FUNCTION_BLOCK MeasurementWidget
VAR_INPUT
    value : LREAL;
    actualStatus : STRING;
END_VAR
VAR_IN_OUT
    healthStatus : HealthStatus;
END_VAR
VAR_OUTPUT
    display : STRING;
    _formatString : FB_FormatString;
END_VAR
VAR
    name : STRING;
    actualStatusWidget : StatusWidget;
    format : STRING;
END_VAR

actualStatusWidget(text  := actualStatus,
                   color := HealthToColor(healthStatus));

IF healthStatus.good OR healthStatus.warning THEN
    _formatString(sFormat := format, 
                  arg1    := F_LREAL(value),
                  sOut    => display);
ELSE
    display := '';
END_IF

METHOD FB_init : BOOL
VAR_INPUT
	bInitRetains : BOOL; // if TRUE, the retain variables are initialized (warm start / cold start)
	bInCopyCode : BOOL;  // if TRUE, the instance afterwards gets moved into the copy code (online change)
    n : STRING;
    f : STRING;
END_VAR
name := n;
format := f;
END_METHOD

END_FUNCTION_BLOCK

(* stored: Version 1.1.0.1, ProductVersion 3.1.4018.2
   POU MeasurementWidget: Id {2fec0466-45e9-42aa-9920-0e9c2cbcfe65}, SpecialFunc None
   Method FB_init: Id {53522e88-6693-469d-835b-729e5c9e25f3} *)
